PROGRAM MAIN
VAR_INPUT
	robot : FB_Robot3R;
	fPosInput : ARRAY [0..2] OF LREAL;
	fVelInput : ARRAY [0..2] OF LREAL;
	
END_VAR
VAR
	bDelayStart : BOOL := FALSE;
	fbDelayStart : TON := (PT := T#2S);
	
	
	
//	t AT %Q* : LREAL;
//	A : ARRAY [0..2] OF LREAL;
//	w : ARRAY [0..2] OF LREAL;
//	TT : ARRAY [0..2] OF LREAL;
//	q_Offset : ARRAY [0..2] OF LREAL;
//	phi_Offset : ARRAY [0..2] OF LREAL;
//	y : ARRAY [0..2] OF LREAL;
//	y_t : ARRAY [0..2] OF LREAL;
	u : ARRAY [0..2] OF LREAL;
	
	j : USINT;
//	i : USINT;
	
	
	timers : ARRAY [0..3] OF TON;
	
	// Task cycle time monitoring
	Ts : LREAL := 0.01;
	fbGetCurrentTaskIdx : GETCURTASKINDEX;
	bCycleTimeExceeded : BOOL;
	nCycleCount : UDINT;

	
	bEStop : BOOL;
	
	bRunStupidRoutine: BOOL;
	
	bVelocityMode : BOOL;
	bPositionMode : BOOL;
	bStop : BOOL;
	
	// IK Data
//	Vt AT %Q* : LREAL := 0.5;
//	radius AT %Q* : LREAL := 0.5;
//	p0 AT %Q* : ARRAY [0..1] OF LREAL := [1.5, 2.5];
//	L  AT %Q* : ARRAY [0..2] OF LREAL := [1.5, 1.5, 1.5];

//	q_t  AT %I* : ARRAY [0..2] OF LREAL;
//	q  AT %I* : ARRAY [0..2] OF LREAL;
	
	
	
//	q_t_DEG : ARRAY [0..2] OF LREAL;
//	q_DEG : ARRAY [0..2] OF LREAL;
	
	deflection : ARRAY [0..2] OF LREAL;
	cumulativeAngle : LREAL;
//	cumulativeVel : LREAL;
	
	//filters
	fbGyroFilters : ARRAY [0..2] OF FB_LowPassFilter;
	fGyroFilterCutoff : ARRAY [0..2] OF LREAL := [ 10.0, 10.0, 10.0 ];
	fLinkGyroVelocity : ARRAY [0..2] OF LREAL;
	stGyroFilterParams : ST_FilterParams;
	bFirstRun : BOOL := TRUE;
	
	// Additive torque based on deflection measurement	
	fShaftAdditiveTorque : ARRAY [0..2] OF LREAL := [0.0, 0.0, 0.0]; // [Nm]
	Kt : ARRAY [0..2] OF LREAL := [0.0, 0.0, 0.0]; // gain for defelectuib compensation
	bEnableDeflectionCompensation : BOOL := FALSE;
	
	//filters for velocity feeback
	fbJointVelFilters : ARRAY [0..2] OF FB_LowPassFilter;
	fJointVelFilterCutoff : ARRAY [0..2] OF LREAL := [ 10.0, 10.0, 10.0 ];
	fElasticOscilationVelocity : ARRAY [0..2] OF LREAL;//differene between joint veocity and velocity measured by gyro
	q_t_Filtered : ARRAY [0..2] OF LREAL;
	stJointVelFilterParams : ST_FilterParams;
	
	

END_VAR

IF bDelayStart THEN
	fbDelayStart(IN := TRUE);
	IF fbDelayStart.Q THEN
		fbDelayStart(IN := FALSE);
		bDelayStart := FALSE;
	END_IF
	RETURN;
END_IF

P_HMI();

stupidRoutine(bRunStupidRoutine:=bRunStupidRoutine);


// Get smaple time from current task
getSampleTime();


IF bFirstRun THEN
	bFirstRun := FALSE;
	FOR j := 0 TO 2 DO
		//initialize Gyro Filters
		stGyroFilterParams.fCutoff := fGyroFilterCutoff[j];
		stGyroFilterParams.fDeltaTime := Ts;
		stGyroFilterParams.fInitialValue := 0.0;
		fbGyroFilters[j].init(stParams := stGyroFilterParams);
		
		//initialize JointVel Filters
		stJointVelFilterParams.fCutoff := fJointVelFilterCutoff[j];
		stJointVelFilterParams.fDeltaTime := Ts;
		stJointVelFilterParams.fInitialValue := 0.0;
		fbJointVelFilters[j].init(stParams := stJointVelFilterParams);
		
	END_FOR
END_IF





cumulativeAngle := 0.0;
//cumulativeVel := 0.0;
FOR j := 0 TO 2 DO
	fbGyroFilters[j].update(IMU.fbStim300[j].ImuData.stGyro.x);
	fLinkGyroVelocity[j] := fbGyroFilters[j].fOut;
	IF j > 0 THEN
		fLinkGyroVelocity[j] := fLinkGyroVelocity[j] - fbGyroFilters[j-1].fOut;
	END_IF
	
	cumulativeAngle := cumulativeAngle + robot.q[j];
	deflection[j] := IMU.fbStim300[j].fRollDegFiltered - cumulativeAngle;
END_FOR


//calculate additive torque
FOR j := 0 TO 2 DO	
	fbJointVelFilters[j].update(robot.q_t[j]);
	q_t_Filtered[j] := fbJointVelFilters[j].fOut;
	fElasticOscilationVelocity[j] := fLinkGyroVelocity[j] - q_t_Filtered[j];
	
	IF bEnableDeflectionCompensation THEN	
		fShaftAdditiveTorque[j] := -Kt[j]*fElasticOscilationVelocity[j];
	ELSE
		fShaftAdditiveTorque[j] := 0.0;	
	END_IF		
END_FOR




robot(
	bEmStop := NOT Safety.TS_I_Safety_EStopOK,
	Ts:=Ts,
	fVelInput:=fVelInput,//u
	fPosInput := fPosInput,
	fShaftAdditiveTorque := fShaftAdditiveTorque,
	fJointPositionOffset := Parameters.fJointPositionOffset,
	fJointCalibrationOffset := Parameters.fJointCalibrationOffset
);

ACTION getSampleTime:
// Get sample time of current task
fbGetCurrentTaskIdx();
bCycleTimeExceeded := _TaskInfo[fbGetCurrentTaskIdx.index].CycleTimeExceeded;
nCycleCount := _TaskInfo[fbGetCurrentTaskIdx.index].CycleCount;
Ts := UDINT_TO_LREAL(_TaskInfo[fbGetCurrentTaskIdx.index].CycleTime/10)/1E6;
END_ACTION

METHOD stupidRoutine : BOOL
VAR_INPUT
	bRunStupidRoutine: BOOL;
END_VAR
timers[0](
	IN:=bRunStupidRoutine,
	PT:=T#2S
);

IF timers[0].Q THEN
	Safety.TS_Q_Safety_GroupPort_ErrAck := TRUE;
	
	timers[1](
		IN:=bRunStupidRoutine,
		PT:=T#1S
	);
	
	IF timers[1].Q THEN
		Safety.TS_Q_Safety_GroupPort_ErrAck := FALSE;
		Safety.TS_Q_Safety_EStopRestart := TRUE;
		
		timers[2](
			IN:=bRunStupidRoutine,
			PT:=T#1S
		);
		
		IF timers[2].Q THEN
			Safety.TS_Q_Safety_EStopRestart := FALSE;
			Safety.TS_Q_Safety_Drive_Axis_ErrReset := TRUE;
			
			timers[3](
				IN:=bRunStupidRoutine,
				PT:=T#1S
			);
			
			IF timers[3].Q THEN
				Safety.TS_Q_Safety_Drive_Axis_ErrReset := FALSE;
				
			END_IF
			
		END_IF
		
	END_IF
	
END_IF
END_METHOD

END_PROGRAM

(* stored: Version 1.1.0.1, ProductVersion 3.1.4024.9
   POU MAIN: Id {870836e7-c1db-4c5e-9373-286a0440b8b4}, SpecialFunc None
   Action getSampleTime: Id {503be4e8-d825-4f62-bfd8-9f7ff9c902be}
   Method stupidRoutine: Id {c599bf63-7edb-4afa-8510-dcae936441fa} *)
